(* PLC project SafeLOGIC-1, BrAutomation SafeDESIGNER  5.15.0.0 *)
(* stored: companyURL http://www.br-automation.com, creationDateTime Thu Jan 05 12:19:48 2023 *)

PROGRAM SafeModuleOk
  VAR  (* added by the conversion: wires and edge detectors of the diagram *)
    _AND_S3_OUT : ANY;
  END_VAR

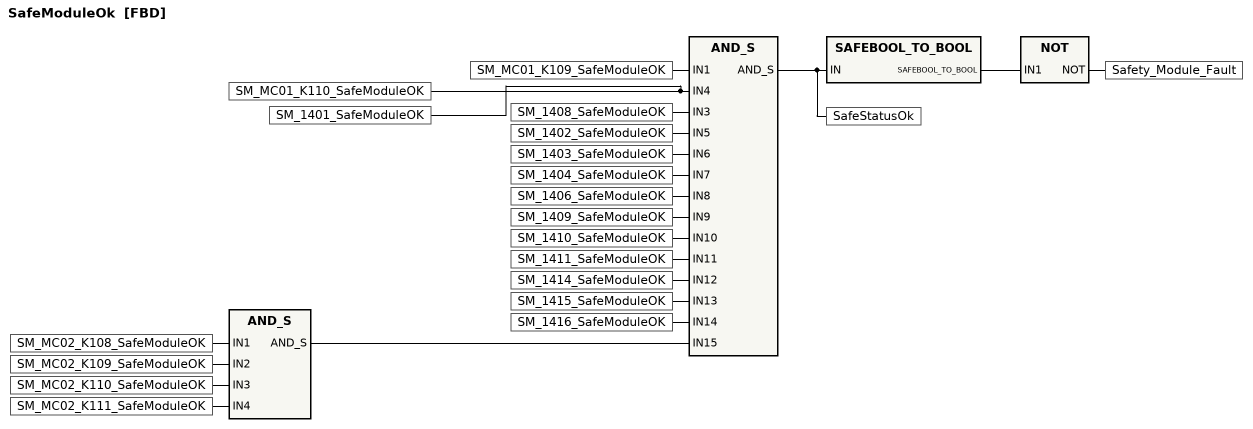
(* FBD diagram, written out as Structured Text *)
_AND_S3_OUT := AND_S(SM_MC01_K109_SafeModuleOK, SM_MC01_K110_SafeModuleOK, SM_1408_SafeModuleOK, SM_1401_SafeModuleOK, SM_1402_SafeModuleOK, SM_1403_SafeModuleOK, SM_1404_SafeModuleOK, SM_1406_SafeModuleOK, SM_1409_SafeModuleOK, SM_1410_SafeModuleOK, SM_1411_SafeModuleOK, SM_1414_SafeModuleOK, SM_1415_SafeModuleOK, SM_1416_SafeModuleOK, AND_S(SM_MC02_K108_SafeModuleOK, SM_MC02_K109_SafeModuleOK, SM_MC02_K110_SafeModuleOK, SM_MC02_K111_SafeModuleOK));
SafeStatusOk := _AND_S3_OUT;
Safety_Module_Fault := NOT SAFEBOOL_TO_BOOL(_AND_S3_OUT);
END_PROGRAM
